{attribute 'GeneratedUsingTerminal: EL9186--0000'}
{attribute addProperty BoxType "EL9186--0000"}
{attribute addProperty Description "EL9186 Potential Connection, 8 x 24V"}
{attribute addProperty Physics "KK"}
{attribute addProperty Id "EL9186"}
{attribute addProperty CRC "2442347326"}
{attribute addProperty Size "0"}
TYPE EL9186_9193433E EXTENDS EtcSlaveTerminalBase_947E5A46 :
STRUCT
END_STRUCT
END_TYPE

(* stored: Version 1.2.0.0, ProductVersion 3.1.4024.11
   DUT EL9186_9193433E: Id {1d7685fe-ef8a-4488-8e87-e329ef1e264b} *)
